FUNCTION_BLOCK T_Parent1 
VAR_INPUT
END_VAR
VAR_OUTPUT
END_VAR
VAR_STAT
	Counter : T_Counter;
END_VAR
VAR

    Child1 : T_Child(Counter, 10);
    Child2 : T_Child(Counter, 20);
    Child3 : T_Child(Counter, 30);
//    Child4 : T_Child(Counter, 1);
END_VAR

METHOD FB_exit : BOOL
VAR_INPUT
	bInCopyCode : BOOL; // if TRUE, the exit method is called for exiting an instance that is copied afterwards (online change).
END_VAR
Counter.Reset();
END_METHOD

END_FUNCTION_BLOCK

(* stored: Version 1.1.0.1, ProductVersion 3.1.4024.12
   POU T_Parent1: Id {8af0ac86-0014-4626-9a27-7de0dee8c9c8}, SpecialFunc None
   Method FB_exit: Id {0170fb1a-b12e-4aa1-8baf-9873b8f5e7aa} *)
